% RSLogix 500 project ALCIP.RSS, saved by version 8.10.00.18 %
PROJECT "ALCIP"    % processor: SLC 500, 1747-L543 %

PROGRAM FILES
  LAD 2   43 rungs
  LAD 3   9 rungs
  LAD 4   18 rungs
  LAD 7   10 rungs
  LAD 8   7 rungs
  LAD 11   60 rungs
  LAD 13   19 rungs
  LAD 15   13 rungs
  LAD 16   17 rungs
  LAD 17   71 rungs
  LAD 18   20 rungs
  LAD 19   20 rungs
  LAD 20   12 rungs
  LAD 21   40 rungs
  LAD 31   74 rungs
  LAD 32   51 rungs
  LAD 33   23 rungs
  LAD 37   92 rungs
  LAD 38   10 rungs
  LAD 39   21 rungs
  LAD 40   16 rungs
  LAD 41   165 rungs
  LAD 42   87 rungs
  LAD 43   5 rungs
  LAD 44   130 rungs
  LAD 45   109 rungs
  LAD 50   39 rungs
  LAD 51   66 rungs
  LAD 52   64 rungs
  LAD 53   84 rungs
  LAD 71   9 rungs
  LAD 74   9 rungs
  LAD 75   28 rungs
  LAD 76   4 rungs
  LAD 77   6 rungs
  LAD 78   2 rungs
  LAD 79   2 rungs
  LAD 80   4 rungs
  LAD 81   2 rungs
  LAD 82   6 rungs
  LAD 83   7 rungs
  LAD 101   33 rungs
  LAD 102   36 rungs
  LAD 70: only END

DATA FILES
  O0 OUTPUT  52 elements
  I1 INPUT  51 elements
  S2 STATUS  164 elements
  B3 BINARY  18 elements
  T4 TIMER  39 elements
  C5 COUNTER  6 elements
  R6 CONTROL  21 elements
  N7 INTEGER  135 elements
  F8 FLOAT  4 elements
  B9   2 elements
  T10   4 elements
  N11   240 elements
  N12   55 elements
  N14   212 elements
  N15   212 elements
  N16   212 elements
  N17   212 elements
  N18   212 elements
  N19   212 elements
  N20   212 elements
  N21   212 elements
  N22   212 elements
  N23   212 elements
  N24   212 elements
  B25   13 elements
  N28   201 elements
  N29   210 elements
  N38   250 elements
  N39   250 elements
  N40   250 elements
  N41   250 elements
  N42   80 elements
  N43   200 elements
  N44   200 elements
  N45   200 elements
  N46   200 elements
  N47   200 elements
  N48   200 elements
  N49   200 elements
  N50   200 elements
  N60   250 elements
  N61   250 elements
  N62   80 elements
  N63   200 elements
  N64   200 elements
  N65   200 elements
  N66   200 elements
  N67   200 elements
  N68   200 elements
  N69   200 elements
  N70   200 elements
  N80   250 elements
  N81   250 elements
  N82   80 elements
  N83   200 elements
  N84   200 elements
  N85   200 elements
  N86   200 elements
  N87   200 elements
  N88   200 elements
  N89   200 elements
  N90   200 elements
  N100   250 elements
  N101   250 elements
  N102   80 elements
  N103   200 elements
  N104   200 elements
  N105   200 elements
  N106   200 elements
  N107   200 elements
  N108   200 elements
  N109   200 elements
  N110   200 elements
  N120   250 elements
  N121   250 elements
  N122   80 elements
  N123   200 elements
  N124   200 elements
  N125   200 elements
  N126   200 elements
  N127   200 elements
  N128   200 elements
  N129   200 elements
  N130   200 elements
  N140   250 elements
  N141   250 elements
  N142   80 elements
  N143   200 elements
  N144   200 elements
  N145   200 elements
  N146   200 elements
  N147   200 elements
  N148   200 elements
  N149   200 elements
  N150   200 elements
  B160   21 elements
  B161   69 elements
  B162   69 elements
  B163   69 elements
  B164   69 elements
  B165   69 elements
  B166   69 elements
  B169   69 elements
  N170   217 elements
  N171   238 elements
  N172   238 elements
  N173   238 elements
  N174   238 elements
  N175   238 elements
  N176   238 elements
  N179   238 elements
  T180   10 elements
  T181   67 elements
  T182   67 elements
  T183   67 elements
  T184   67 elements
  T185   67 elements
  T186   67 elements
  N191   80 elements
  N192   80 elements
  N193   80 elements
  N194   80 elements
  N195   80 elements
  N196   80 elements
  N200   131 elements
  N201   17 elements
  N202   17 elements
  N203   17 elements
  N204   17 elements
  N205   17 elements
  N206   17 elements
  N210   43 elements
  N211   43 elements
  N212   43 elements
  N213   43 elements
  N214   43 elements
  N215   43 elements
  N216   43 elements
  N220   250 elements
  N221   250 elements
  N231   73 elements
  N232   73 elements
  N233   73 elements
  N234   73 elements
  N235   73 elements
  N236   73 elements

LADDER 2
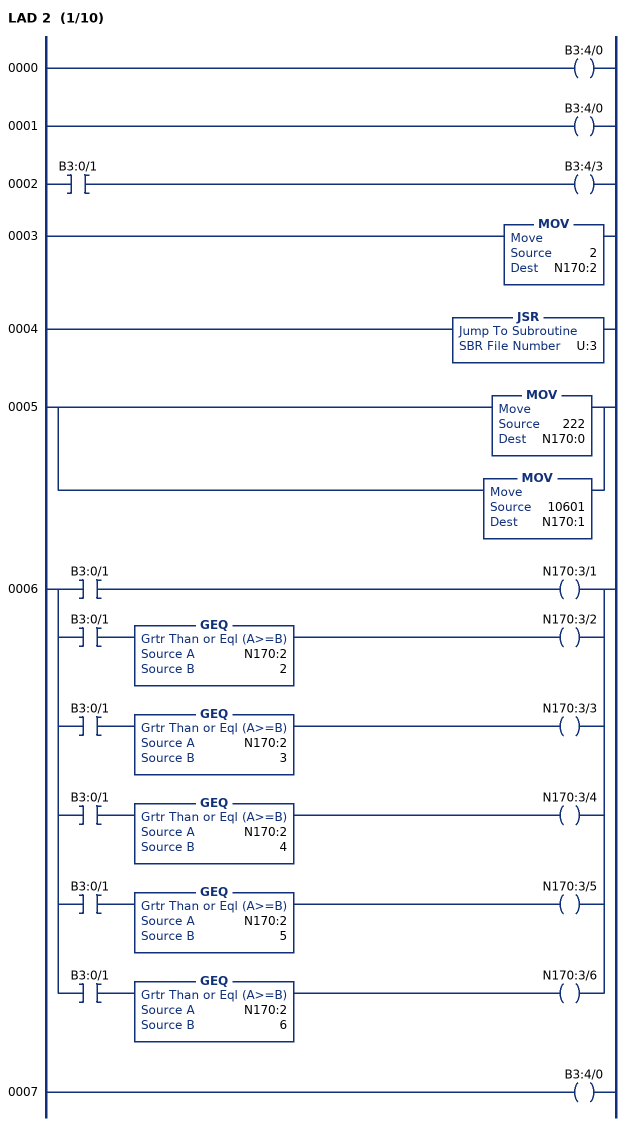
% Rung: 0 %
SOR OTE B3:4/0 EOR
% Rung: 1 %
SOR OTE B3:4/0 EOR
% Rung: 2 %
SOR XIC B3:0/1 OTE B3:4/3 EOR
% Rung: 3 %
SOR MOV 2 N170:2 EOR
% Rung: 4 %
SOR JSR U:3 EOR
% Rung: 5 %
SOR BST MOV 222 N170:0 NXB MOV 10601 N170:1 BND EOR
% Rung: 6 %
SOR BST XIC B3:0/1 OTE N170:3/1 NXB XIC B3:0/1 GEQ N170:2 2 OTE N170:3/2 NXB XIC B3:0/1 GEQ N170:2 3 OTE N170:3/3 NXB XIC B3:0/1 GEQ N170:2 4 OTE N170:3/4 NXB XIC B3:0/1 GEQ N170:2 5 OTE N170:3/5 NXB XIC B3:0/1 GEQ N170:2 6 OTE N170:3/6 BND EOR
% Rung: 7 %
SOR OTE B3:4/0 EOR

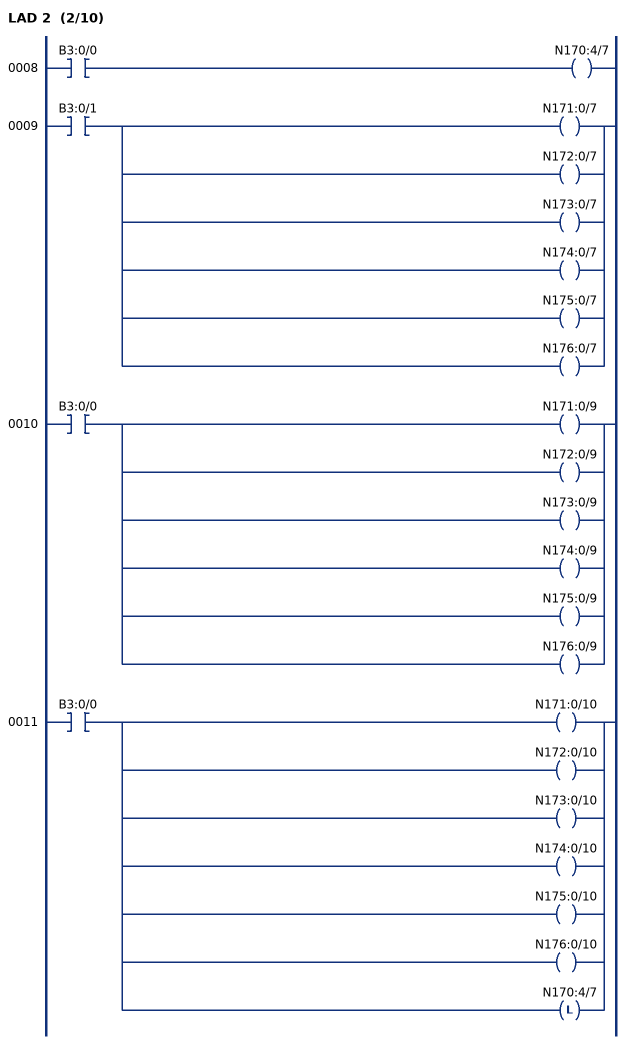
% Rung: 8 %
SOR XIC B3:0/0 OTE N170:4/7 EOR
% Rung: 9 %
SOR XIC B3:0/1 BST OTE N171:0/7 NXB OTE N172:0/7 NXB OTE N173:0/7 NXB OTE N174:0/7 NXB OTE N175:0/7 NXB OTE N176:0/7 BND EOR
% Rung: 10 %
SOR XIC B3:0/0 BST OTE N171:0/9 NXB OTE N172:0/9 NXB OTE N173:0/9 NXB OTE N174:0/9 NXB OTE N175:0/9 NXB OTE N176:0/9 BND EOR
% Rung: 11 %
SOR XIC B3:0/0 BST BST OTE N171:0/10 NXB OTE N172:0/10 NXB OTE N173:0/10 NXB OTE N174:0/10 NXB OTE N175:0/10 NXB OTE N176:0/10 BND NXB OTL N170:4/7 BND EOR

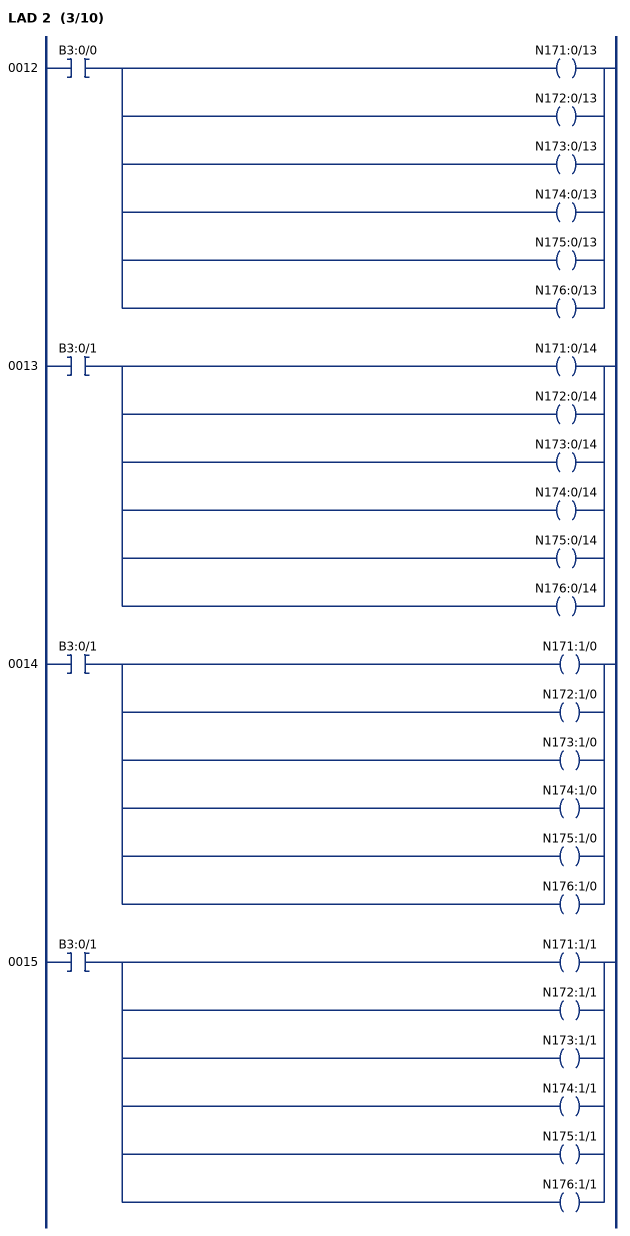
% Rung: 12 %
SOR XIC B3:0/0 BST OTE N171:0/13 NXB OTE N172:0/13 NXB OTE N173:0/13 NXB OTE N174:0/13 NXB OTE N175:0/13 NXB OTE N176:0/13 BND EOR
% Rung: 13 %
SOR XIC B3:0/1 BST OTE N171:0/14 NXB OTE N172:0/14 NXB OTE N173:0/14 NXB OTE N174:0/14 NXB OTE N175:0/14 NXB OTE N176:0/14 BND EOR
% Rung: 14 %
SOR XIC B3:0/1 BST OTE N171:1/0 NXB OTE N172:1/0 NXB OTE N173:1/0 NXB OTE N174:1/0 NXB OTE N175:1/0 NXB OTE N176:1/0 BND EOR
% Rung: 15 %
SOR XIC B3:0/1 BST OTE N171:1/1 NXB OTE N172:1/1 NXB OTE N173:1/1 NXB OTE N174:1/1 NXB OTE N175:1/1 NXB OTE N176:1/1 BND EOR

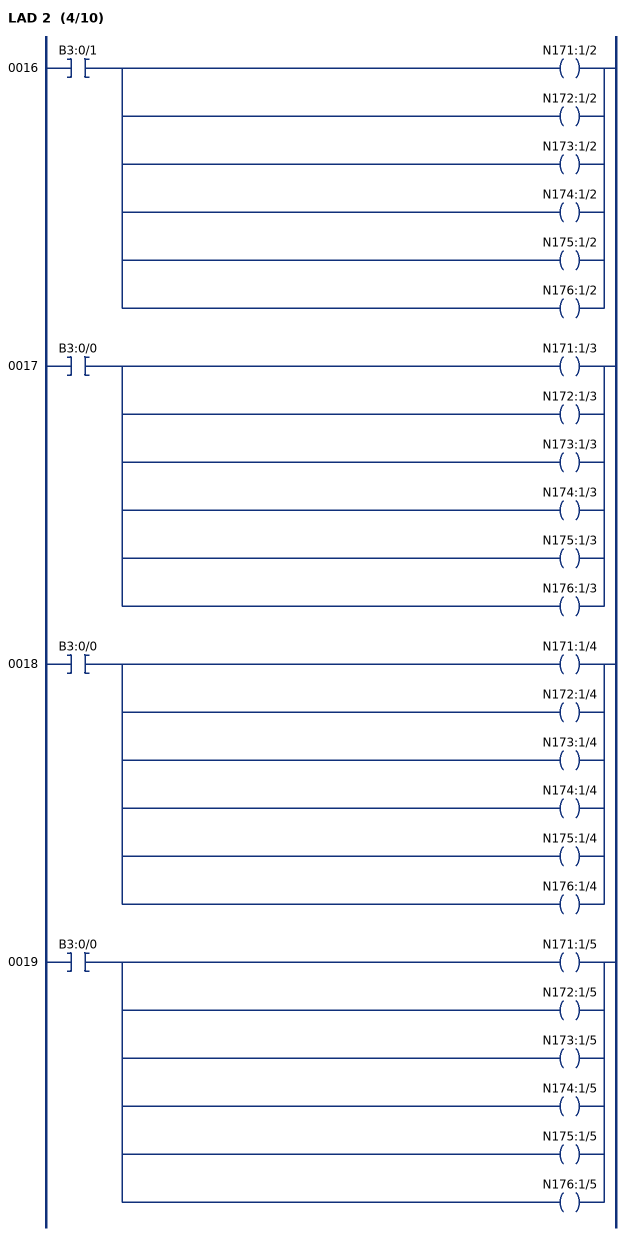
% Rung: 16 %
SOR XIC B3:0/1 BST OTE N171:1/2 NXB OTE N172:1/2 NXB OTE N173:1/2 NXB OTE N174:1/2 NXB OTE N175:1/2 NXB OTE N176:1/2 BND EOR
% Rung: 17 %
SOR XIC B3:0/0 BST OTE N171:1/3 NXB OTE N172:1/3 NXB OTE N173:1/3 NXB OTE N174:1/3 NXB OTE N175:1/3 NXB OTE N176:1/3 BND EOR
% Rung: 18 %
SOR XIC B3:0/0 BST OTE N171:1/4 NXB OTE N172:1/4 NXB OTE N173:1/4 NXB OTE N174:1/4 NXB OTE N175:1/4 NXB OTE N176:1/4 BND EOR
% Rung: 19 %
SOR XIC B3:0/0 BST OTE N171:1/5 NXB OTE N172:1/5 NXB OTE N173:1/5 NXB OTE N174:1/5 NXB OTE N175:1/5 NXB OTE N176:1/5 BND EOR

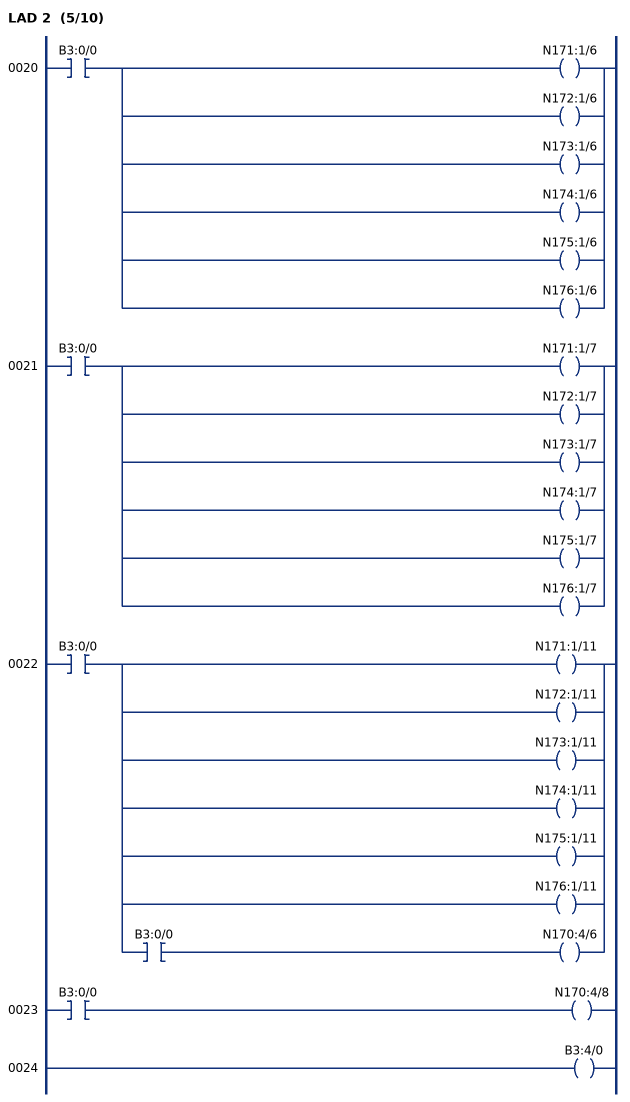
% Rung: 20 %
SOR XIC B3:0/0 BST OTE N171:1/6 NXB OTE N172:1/6 NXB OTE N173:1/6 NXB OTE N174:1/6 NXB OTE N175:1/6 NXB OTE N176:1/6 BND EOR
% Rung: 21 %
SOR XIC B3:0/0 BST OTE N171:1/7 NXB OTE N172:1/7 NXB OTE N173:1/7 NXB OTE N174:1/7 NXB OTE N175:1/7 NXB OTE N176:1/7 BND EOR
% Rung: 22 %
SOR XIC B3:0/0 BST OTE N171:1/11 NXB OTE N172:1/11 NXB OTE N173:1/11 NXB OTE N174:1/11 NXB OTE N175:1/11 NXB OTE N176:1/11 NXB XIC B3:0/0 OTE N170:4/6 BND EOR
% Rung: 23 %
SOR XIC B3:0/0 OTE N170:4/8 EOR
% Rung: 24 %
SOR OTE B3:4/0 EOR

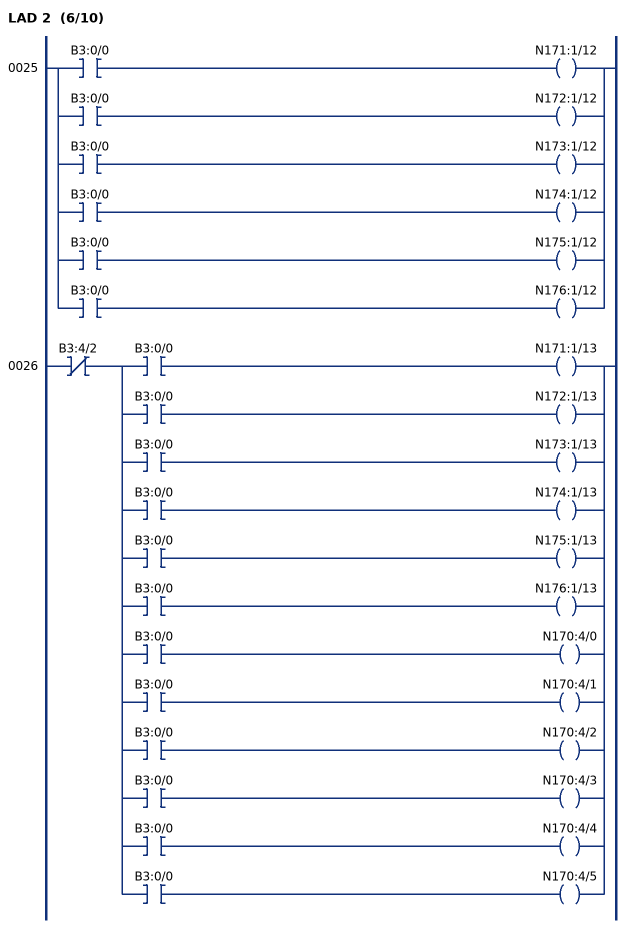
% Rung: 25 %
SOR BST XIC B3:0/0 OTE N171:1/12 NXB XIC B3:0/0 OTE N172:1/12 NXB XIC B3:0/0 OTE N173:1/12 NXB XIC B3:0/0 OTE N174:1/12 NXB XIC B3:0/0 OTE N175:1/12 NXB XIC B3:0/0 OTE N176:1/12 BND EOR
% Rung: 26 %
SOR XIO B3:4/2 BST BST XIC B3:0/0 OTE N171:1/13 NXB XIC B3:0/0 OTE N172:1/13 NXB XIC B3:0/0 OTE N173:1/13 NXB XIC B3:0/0 OTE N174:1/13 NXB XIC B3:0/0 OTE N175:1/13 NXB XIC B3:0/0 OTE N176:1/13 BND NXB XIC B3:0/0 OTE N170:4/0 NXB XIC B3:0/0 OTE N170:4/1 NXB XIC B3:0/0 OTE N170:4/2 NXB XIC B3:0/0 OTE N170:4/3 NXB XIC B3:0/0 OTE N170:4/4 NXB XIC B3:0/0 OTE N170:4/5 BND EOR

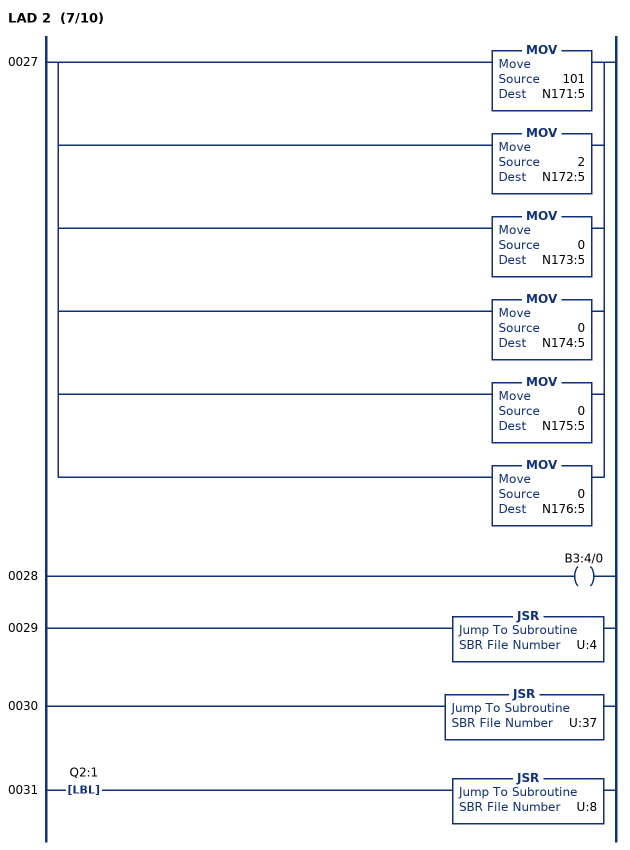
% Rung: 27 %
SOR BST MOV 101 N171:5 NXB MOV 2 N172:5 NXB MOV 0 N173:5 NXB MOV 0 N174:5 NXB MOV 0 N175:5 NXB MOV 0 N176:5 BND EOR
% Rung: 28 %
SOR OTE B3:4/0 EOR
% Rung: 29 %
SOR JSR U:4 EOR
% Rung: 30 %
SOR JSR U:37 EOR
% Rung: 31 %
SOR LBL Q2:1 JSR U:8 EOR

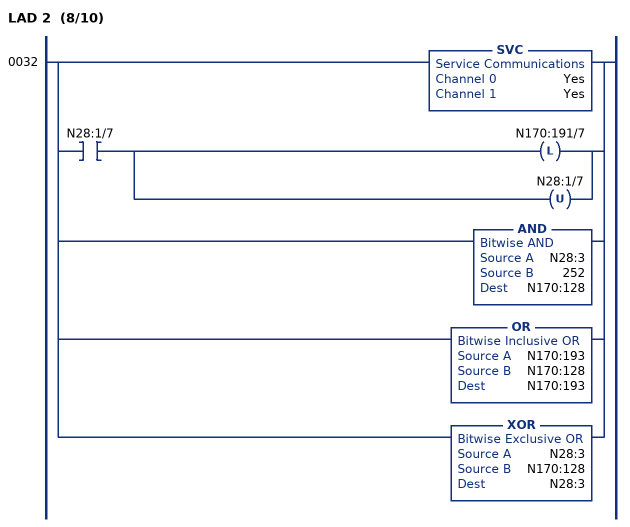
% Rung: 32 %
SOR BST SVC Yes Yes NXB XIC N28:1/7 BST OTL N170:191/7 NXB OTU N28:1/7 BND NXB AND N28:3 252 N170:128 NXB OR N170:193 N170:128 N170:193 NXB XOR N28:3 N170:128 N28:3 BND EOR

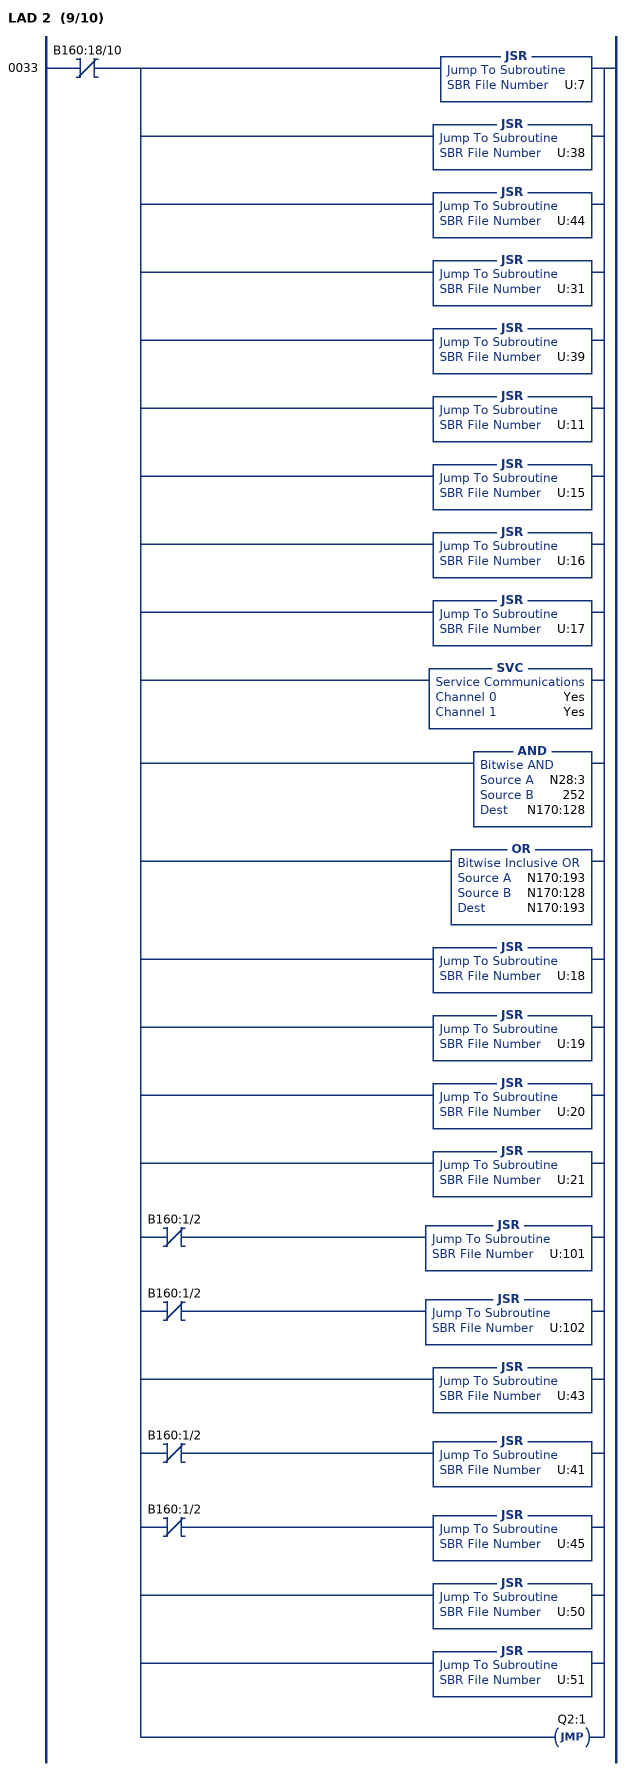
% Rung: 33 %
SOR XIO B160:18/10 BST JSR U:7 NXB JSR U:38 NXB JSR U:44 NXB JSR U:31 NXB JSR U:39 NXB JSR U:11 NXB JSR U:15 NXB JSR U:16 NXB JSR U:17 NXB BST SVC Yes Yes NXB AND N28:3 252 N170:128 NXB OR N170:193 N170:128 N170:193 BND NXB JSR U:18 NXB JSR U:19 NXB JSR U:20 NXB JSR U:21 NXB XIO B160:1/2 JSR U:101 NXB XIO B160:1/2 JSR U:102 NXB JSR U:43 NXB XIO B160:1/2 JSR U:41 NXB XIO B160:1/2 JSR U:45 NXB JSR U:50 NXB JSR U:51 NXB JMP Q2:1 BND EOR

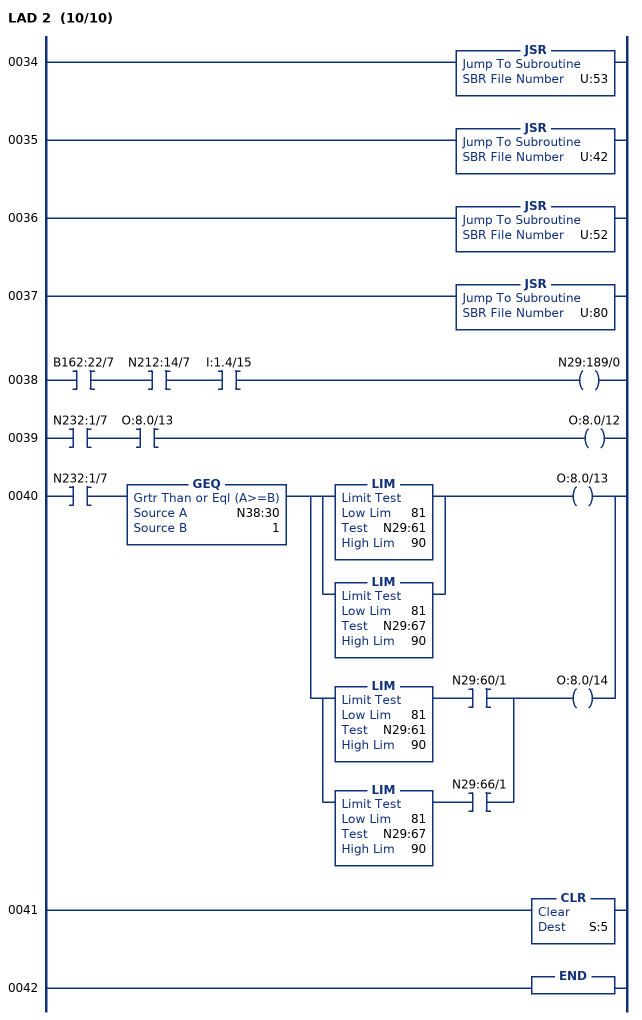
% Rung: 34 %
SOR JSR U:53 EOR
% Rung: 35 %
SOR JSR U:42 EOR
% Rung: 36 %
SOR JSR U:52 EOR
% Rung: 37 %
SOR JSR U:80 EOR
% Rung: 38 %
SOR XIC B162:22/7 XIC N212:14/7 XIC I:1.4/15 OTE N29:189/0 EOR
% Rung: 39 %
SOR XIC N232:1/7 XIC O:8.0/13 OTE O:8.0/12 EOR
% Rung: 40 %
SOR XIC N232:1/7 GEQ N38:30 1 BST BST LIM 81 N29:61 90 NXB LIM 81 N29:67 90 BND OTE O:8.0/13 NXB BST LIM 81 N29:61 90 XIC N29:60/1 NXB LIM 81 N29:67 90 XIC N29:66/1 BND OTE O:8.0/14 BND EOR
% Rung: 41 %
SOR CLR S:5 EOR
% Rung: 42 %
SOR END EOR

LADDER 3
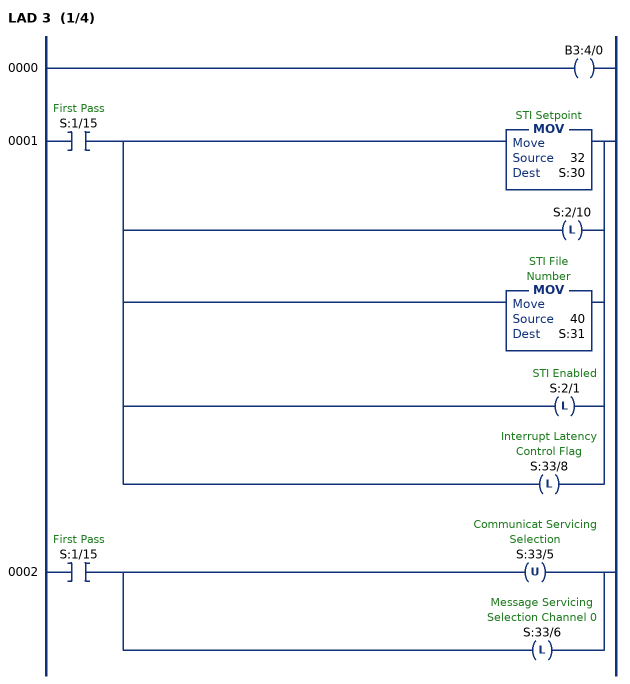
% Rung: 0 %
SOR OTE B3:4/0 EOR
% Rung: 1 %
SOR XIC S:1/15 BST MOV 32 S:30 NXB OTL S:2/10 NXB MOV 40 S:31 NXB OTL S:2/1 NXB OTL S:33/8 BND EOR
%   S:1/15  "First Pass" %
%   S:30  "STI Setpoint" %
%   S:31  "STI File Number" %
%   S:2/1  "STI Enabled" %
%   S:33/8  "Interrupt Latency Control Flag" %
% Rung: 2 %
SOR XIC S:1/15 BST OTU S:33/5 NXB OTL S:33/6 BND EOR
%   S:1/15  "First Pass" %
%   S:33/5  "Communicat Servicing Selection" %
%   S:33/6  "Message Servicing Selection Channel 0" %

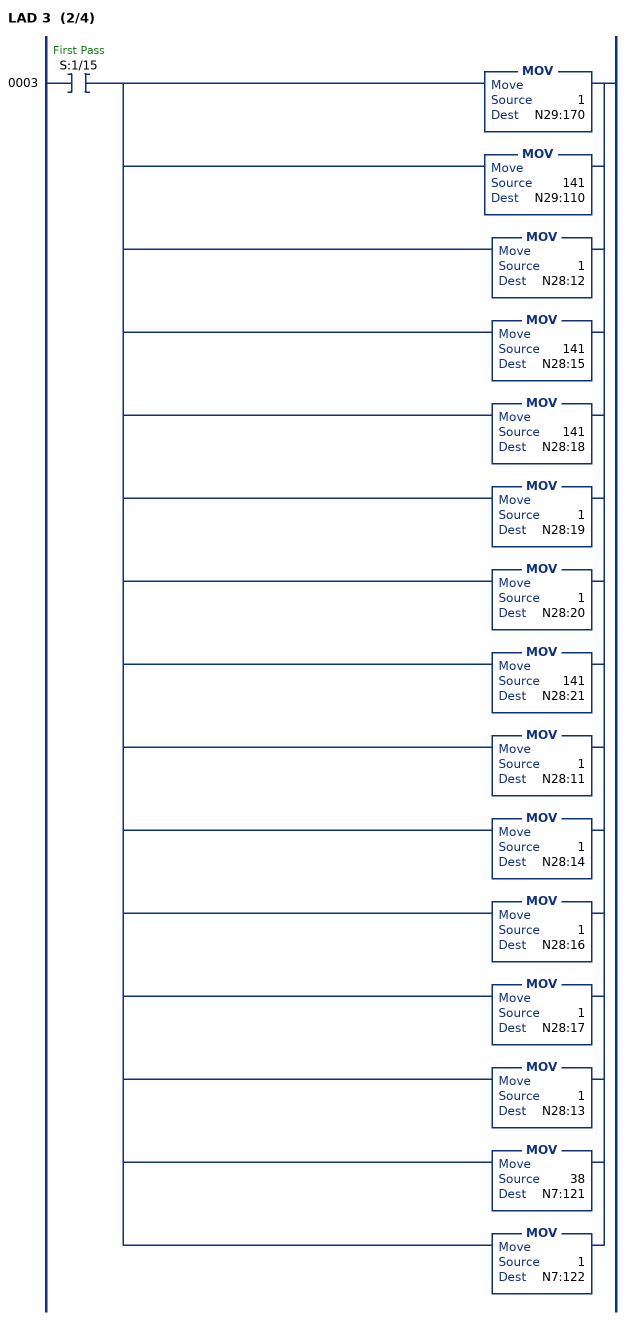
% Rung: 3 %
SOR XIC S:1/15 BST MOV 1 N29:170 NXB MOV 141 N29:110 NXB MOV 1 N28:12 NXB MOV 141 N28:15 NXB MOV 141 N28:18 NXB MOV 1 N28:19 NXB MOV 1 N28:20 NXB MOV 141 N28:21 NXB MOV 1 N28:11 NXB MOV 1 N28:14 NXB MOV 1 N28:16 NXB MOV 1 N28:17 NXB MOV 1 N28:13 NXB MOV 38 N7:121 NXB MOV 1 N7:122 BND EOR
%   S:1/15  "First Pass" %

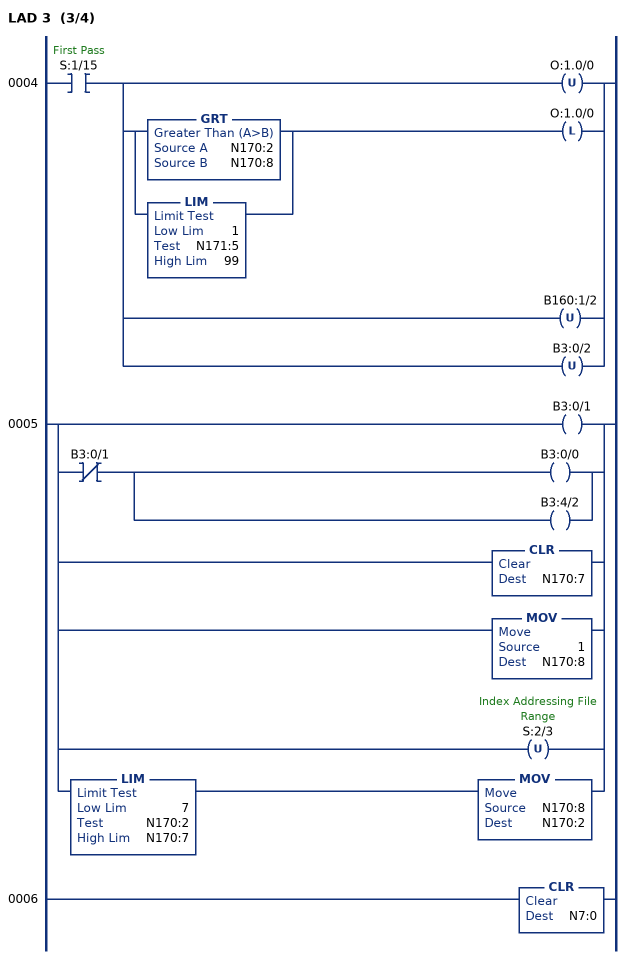
% Rung: 4 %
SOR XIC S:1/15 BST BST OTU O:1.0/0 NXB BST GRT N170:2 N170:8 NXB LIM 1 N171:5 99 BND OTL O:1.0/0 BND NXB OTU B160:1/2 NXB OTU B3:0/2 BND EOR
%   S:1/15  "First Pass" %
% Rung: 5 %
SOR BST OTE B3:0/1 NXB XIO B3:0/1 BST OTE B3:0/0 NXB OTE B3:4/2 BND NXB CLR N170:7 NXB MOV 1 N170:8 NXB OTU S:2/3 NXB LIM 7 N170:2 N170:7 MOV N170:8 N170:2 BND EOR
%   S:2/3  "Index Addressing File Range" %
% Rung: 6 %
SOR CLR N7:0 EOR

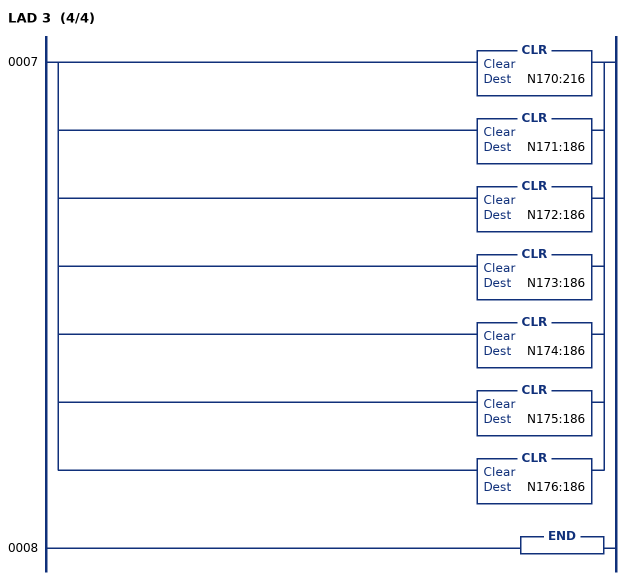
% Rung: 7 %
SOR BST CLR N170:216 NXB CLR N171:186 NXB CLR N172:186 NXB CLR N173:186 NXB CLR N174:186 NXB CLR N175:186 NXB CLR N176:186 BND EOR
% Rung: 8 %
SOR END EOR

LADDER 4
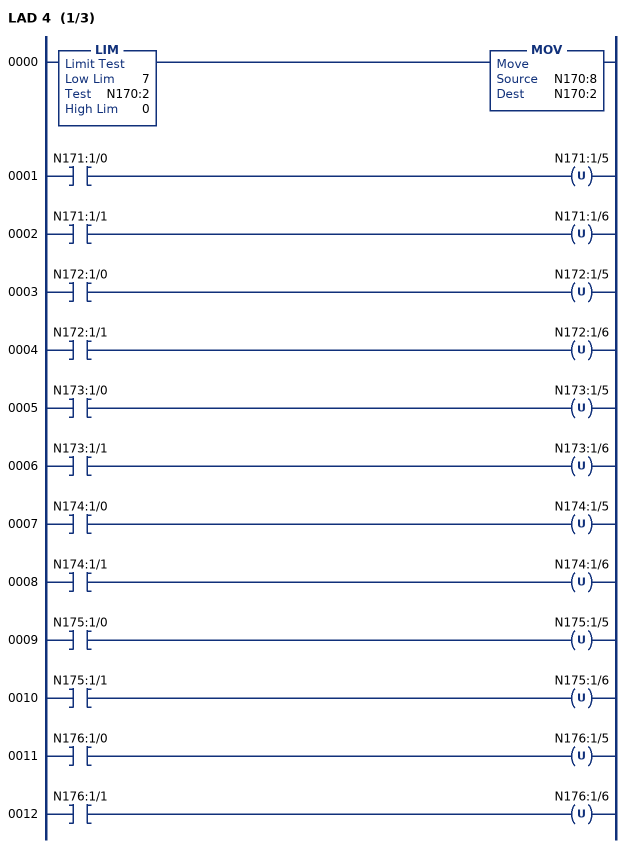
% Rung: 0 %
SOR LIM 7 N170:2 0 MOV N170:8 N170:2 EOR
% Rung: 1 %
SOR XIC N171:1/0 OTU N171:1/5 EOR
% Rung: 2 %
SOR XIC N171:1/1 OTU N171:1/6 EOR
% Rung: 3 %
SOR XIC N172:1/0 OTU N172:1/5 EOR
% Rung: 4 %
SOR XIC N172:1/1 OTU N172:1/6 EOR
% Rung: 5 %
SOR XIC N173:1/0 OTU N173:1/5 EOR
% Rung: 6 %
SOR XIC N173:1/1 OTU N173:1/6 EOR
% Rung: 7 %
SOR XIC N174:1/0 OTU N174:1/5 EOR
% Rung: 8 %
SOR XIC N174:1/1 OTU N174:1/6 EOR
% Rung: 9 %
SOR XIC N175:1/0 OTU N175:1/5 EOR
% Rung: 10 %
SOR XIC N175:1/1 OTU N175:1/6 EOR
% Rung: 11 %
SOR XIC N176:1/0 OTU N176:1/5 EOR
% Rung: 12 %
SOR XIC N176:1/1 OTU N176:1/6 EOR

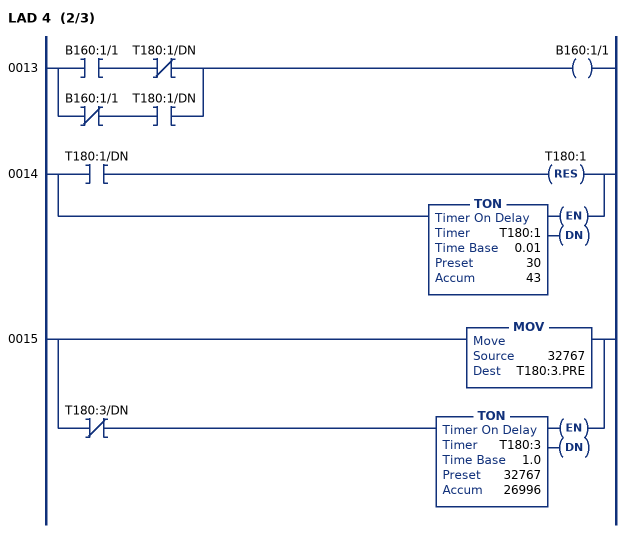
% Rung: 13 %
SOR BST XIC B160:1/1 XIO T180:1/DN NXB XIO B160:1/1 XIC T180:1/DN BND OTE B160:1/1 EOR
% Rung: 14 %
SOR BST XIC T180:1/DN RES T180:1 NXB TON T180:1 0.01 30 43 BND EOR
% Rung: 15 %
SOR BST MOV 32767 T180:3.PRE NXB XIO T180:3/DN TON T180:3 1.0 32767 26996 BND EOR

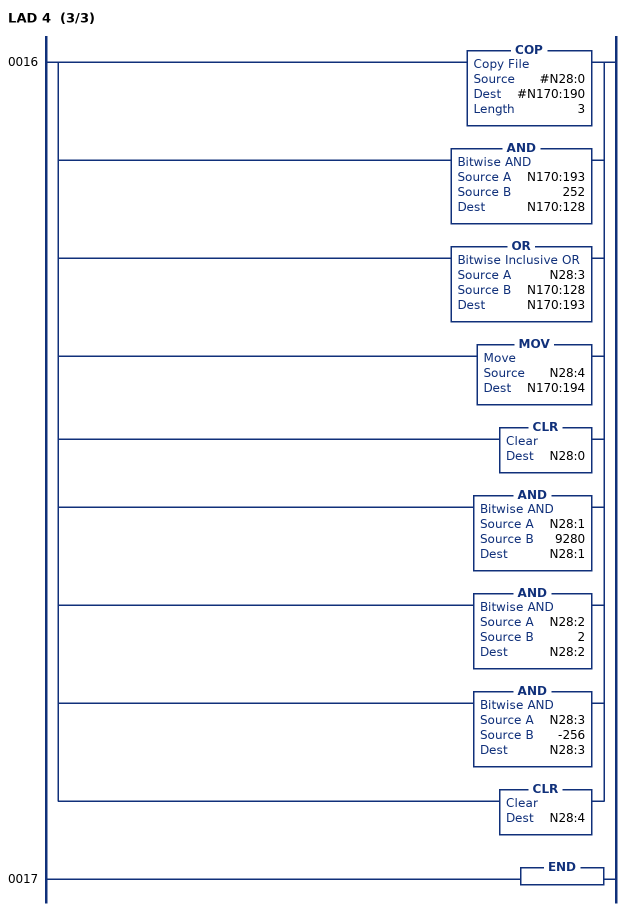
% Rung: 16 %
SOR BST COP #N28:0 #N170:190 3 NXB BST AND N170:193 252 N170:128 NXB OR N28:3 N170:128 N170:193 BND NXB MOV N28:4 N170:194 NXB CLR N28:0 NXB AND N28:1 9280 N28:1 NXB AND N28:2 2 N28:2 NXB AND N28:3 -256 N28:3 NXB CLR N28:4 BND EOR
% Rung: 17 %
SOR END EOR

LADDER 7
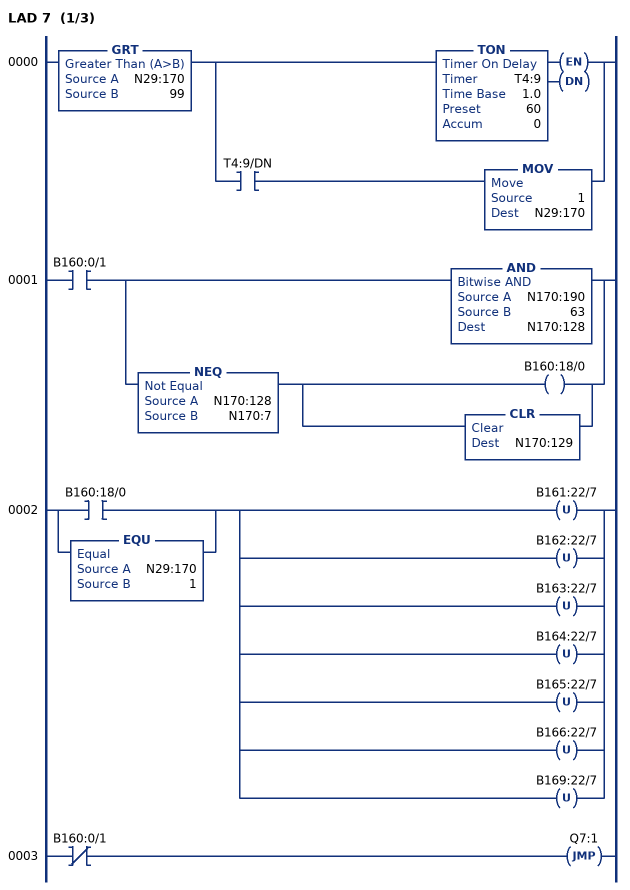
% Rung: 0 %
SOR GRT N29:170 99 BST TON T4:9 1.0 60 0 NXB XIC T4:9/DN MOV 1 N29:170 BND EOR
% Rung: 1 %
SOR XIC B160:0/1 BST AND N170:190 63 N170:128 NXB NEQ N170:128 N170:7 BST OTE B160:18/0 NXB CLR N170:129 BND BND EOR
% Rung: 2 %
SOR BST XIC B160:18/0 NXB EQU N29:170 1 BND BST OTU B161:22/7 NXB OTU B162:22/7 NXB OTU B163:22/7 NXB OTU B164:22/7 NXB OTU B165:22/7 NXB OTU B166:22/7 NXB OTU B169:22/7 BND EOR
% Rung: 3 %
SOR XIO B160:0/1 JMP Q7:1 EOR

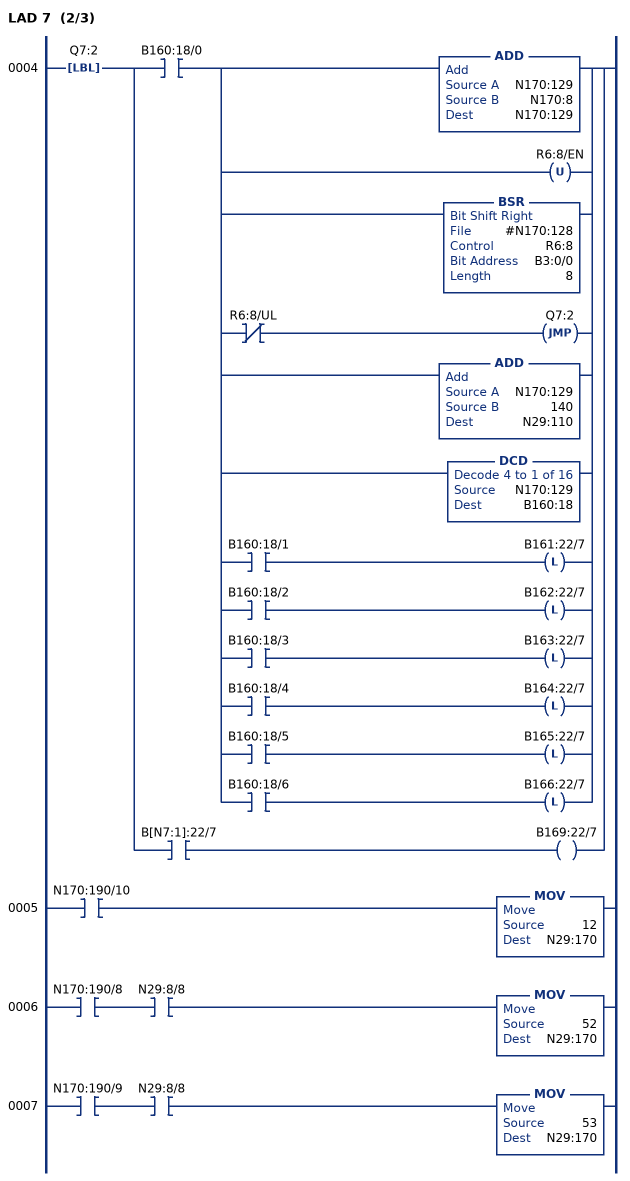
% Rung: 4 %
SOR LBL Q7:2 BST XIC B160:18/0 BST ADD N170:129 N170:8 N170:129 NXB OTU R6:8/EN NXB BSR #N170:128 R6:8 B3:0/0 8 NXB XIO R6:8/UL JMP Q7:2 NXB ADD N170:129 140 N29:110 NXB DCD N170:129 B160:18 NXB XIC B160:18/1 OTL B161:22/7 NXB XIC B160:18/2 OTL B162:22/7 NXB XIC B160:18/3 OTL B163:22/7 NXB XIC B160:18/4 OTL B164:22/7 NXB XIC B160:18/5 OTL B165:22/7 NXB XIC B160:18/6 OTL B166:22/7 BND NXB XIC B[N7:1]:22/7 OTE B169:22/7 BND EOR
% Rung: 5 %
SOR XIC N170:190/10 MOV 12 N29:170 EOR
% Rung: 6 %
SOR XIC N170:190/8 XIC N29:8/8 MOV 52 N29:170 EOR
% Rung: 7 %
SOR XIC N170:190/9 XIC N29:8/8 MOV 53 N29:170 EOR

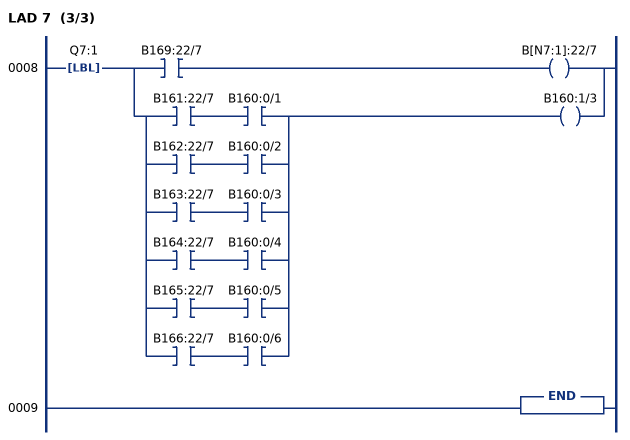
% Rung: 8 %
SOR LBL Q7:1 BST XIC B169:22/7 OTE B[N7:1]:22/7 NXB BST XIC B161:22/7 XIC B160:0/1 NXB XIC B162:22/7 XIC B160:0/2 NXB XIC B163:22/7 XIC B160:0/3 NXB XIC B164:22/7 XIC B160:0/4 NXB XIC B165:22/7 XIC B160:0/5 NXB XIC B166:22/7 XIC B160:0/6 BND OTE B160:1/3 BND EOR
% Rung: 9 %
SOR END EOR

LADDER 8
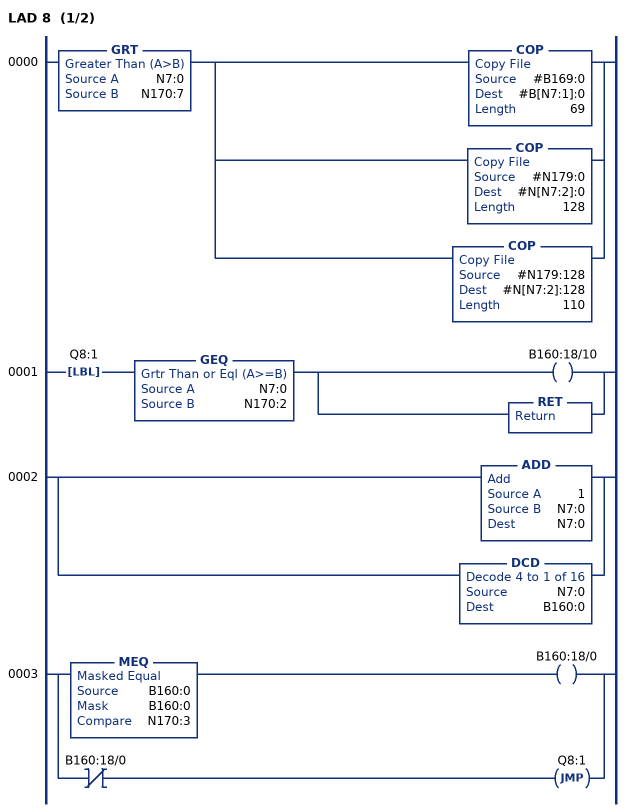
% Rung: 0 %
SOR GRT N7:0 N170:7 BST COP #B169:0 #B[N7:1]:0 69 NXB COP #N179:0 #N[N7:2]:0 128 NXB COP #N179:128 #N[N7:2]:128 110 BND EOR
% Rung: 1 %
SOR LBL Q8:1 GEQ N7:0 N170:2 BST OTE B160:18/10 NXB RET BND EOR
% Rung: 2 %
SOR BST ADD 1 N7:0 N7:0 NXB DCD N7:0 B160:0 BND EOR
% Rung: 3 %
SOR BST MEQ B160:0 B160:0 N170:3 OTE B160:18/0 NXB XIO B160:18/0 JMP Q8:1 BND EOR

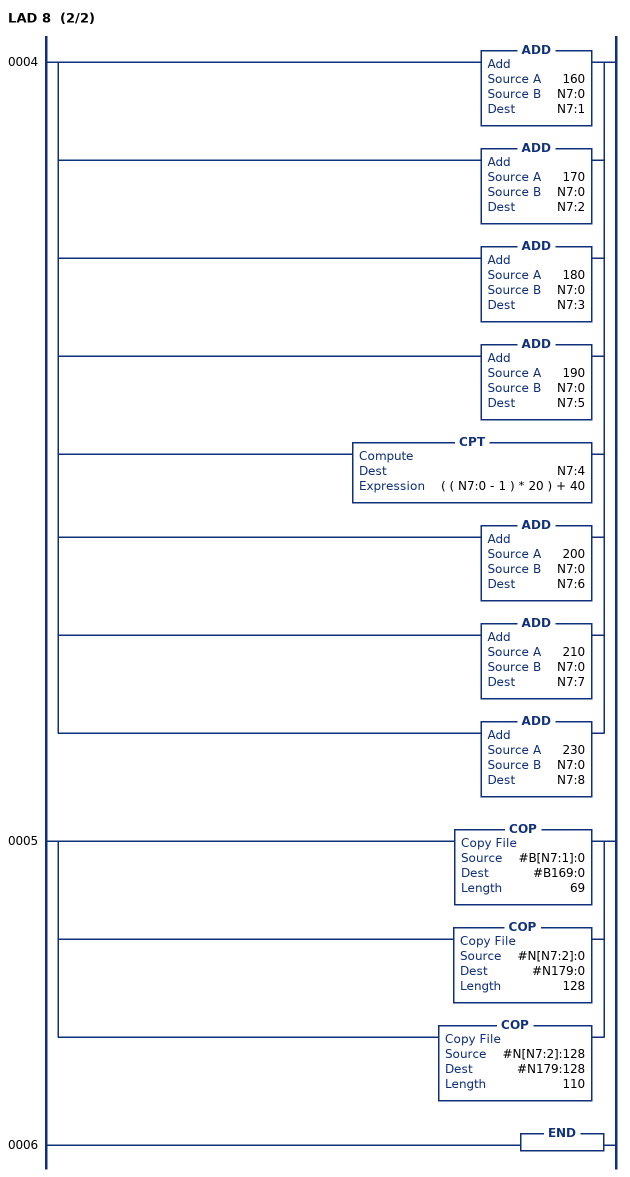
% Rung: 4 %
SOR BST ADD 160 N7:0 N7:1 NXB ADD 170 N7:0 N7:2 NXB ADD 180 N7:0 N7:3 NXB ADD 190 N7:0 N7:5 NXB CPT N7:4 " ( ( N7:0 - 1 ) * 20 ) + 40 " NXB ADD 200 N7:0 N7:6 NXB ADD 210 N7:0 N7:7 NXB ADD 230 N7:0 N7:8 BND EOR
% Rung: 5 %
SOR BST COP #B[N7:1]:0 #B169:0 69 NXB COP #N[N7:2]:0 #N179:0 128 NXB COP #N[N7:2]:128 #N179:128 110 BND EOR
% Rung: 6 %
SOR END EOR

LADDER 11
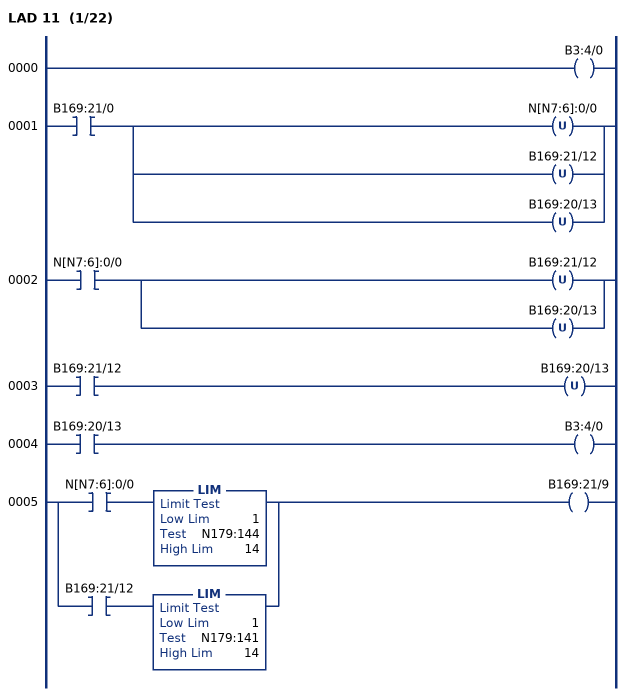
% Rung: 0 %
SOR OTE B3:4/0 EOR
% Rung: 1 %
SOR XIC B169:21/0 BST OTU N[N7:6]:0/0 NXB OTU B169:21/12 NXB OTU B169:20/13 BND EOR
% Rung: 2 %
SOR XIC N[N7:6]:0/0 BST OTU B169:21/12 NXB OTU B169:20/13 BND EOR
% Rung: 3 %
SOR XIC B169:21/12 OTU B169:20/13 EOR
% Rung: 4 %
SOR XIC B169:20/13 OTE B3:4/0 EOR
% Rung: 5 %
SOR BST XIC N[N7:6]:0/0 LIM 1 N179:144 14 NXB XIC B169:21/12 LIM 1 N179:141 14 BND OTE B169:21/9 EOR

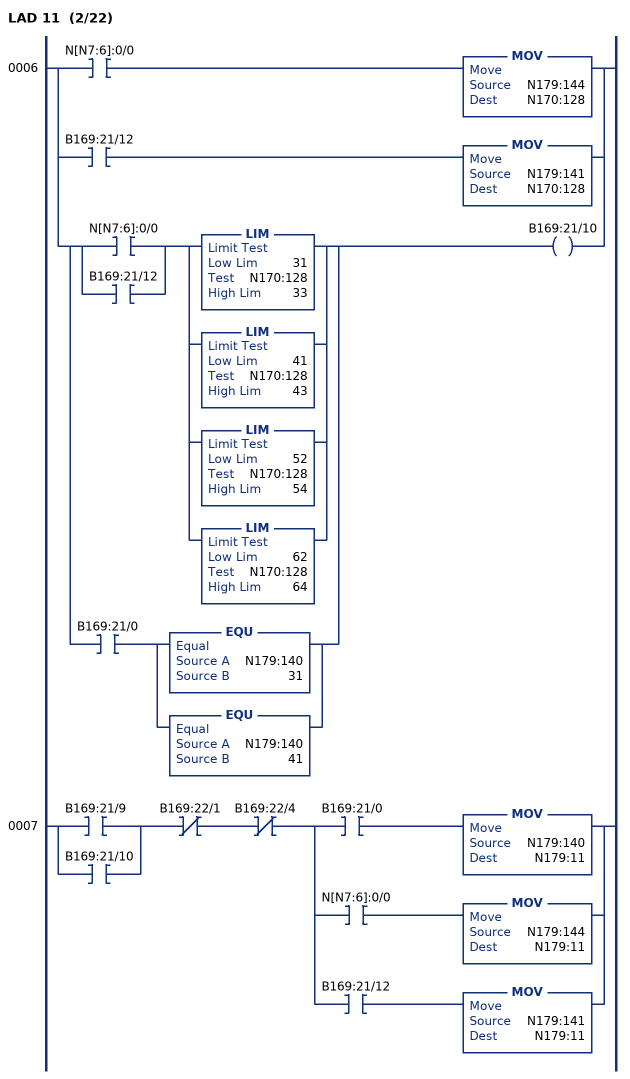
% Rung: 6 %
SOR BST BST XIC N[N7:6]:0/0 MOV N179:144 N170:128 NXB XIC B169:21/12 MOV N179:141 N170:128 BND NXB BST BST XIC N[N7:6]:0/0 NXB XIC B169:21/12 BND BST LIM 31 N170:128 33 NXB LIM 41 N170:128 43 NXB LIM 52 N170:128 54 NXB LIM 62 N170:128 64 BND NXB XIC B169:21/0 BST EQU N179:140 31 NXB EQU N179:140 41 BND BND OTE B169:21/10 BND EOR
% Rung: 7 %
SOR BST XIC B169:21/9 NXB XIC B169:21/10 BND XIO B169:22/1 XIO B169:22/4 BST XIC B169:21/0 MOV N179:140 N179:11 NXB XIC N[N7:6]:0/0 MOV N179:144 N179:11 NXB XIC B169:21/12 MOV N179:141 N179:11 BND EOR

